FUNCTION_BLOCK FB_QueueJobContainerCreator IMPLEMENTS I_TaskCreator
VAR_INPUT
END_VAR
VAR_OUTPUT
END_VAR
VAR
END_VAR

METHOD create_future : I_Future
VAR_INPUT
	future_name	: STRING;
END_VAR
VAR
	_p_future : POINTER TO FB_QueueJobContainer;
END_VAR
_p_future := __NEW(FB_QueueJobContainer);
_p_future^.future_name := future_name;
create_future := _p_future^;
END_METHOD

METHOD destroy_future : I_Future
VAR_INPUT
	future	: I_Future;
END_VAR
VAR
	_p_future : POINTER TO FB_QueueJobContainer;
END_VAR
IF __QUERYPOINTER(future, _p_future) THEN
	__DELETE(_p_future);
	IF _p_future = 0  THEN
		destroy_future := 0;
	END_IF
END_IF
END_METHOD

END_FUNCTION_BLOCK

(* stored: Version 1.1.0.1, ProductVersion 3.1.4026.17
   POU FB_QueueJobContainerCreator: Id {04c4e3d6-d95d-4e06-a90d-cfdc5b2939d5}, SpecialFunc None
   Method create_future: Id {bac6e106-0b4e-45d4-8918-c7e9f3ec886e}
   Method destroy_future: Id {fe84d8ae-214c-473c-b48f-e5e0453688cb} *)
